{attribute 'qualified_only'}
TYPE E_DIAGNOSISTYPE :
(
    InfoMessage := 0,
    WarningMessage := 1,
    ErrorMessage := 2,
    Unspecified := 3
) BYTE;
END_TYPE

(* stored: Version 1.1.0.1, ProductVersion 3.1.4022.12
   DUT E_DIAGNOSISTYPE: Id {9b10da99-659b-4bb5-bdfb-03993909bc0c} *)
